// TIA Portal V17 export
// export: Created 2023-12-22T15:04:44.870563Z, ExportSetting WithDefaults, DisplayName Totally Integrated Automation Portal, DisplayVersion V17, DisplayName TIA Portal Openness, DisplayVersion V17, DisplayName TIA Portal Version Control Interface, DisplayVersion V17, DisplayName STEP 7 Professional, DisplayVersion V17, DisplayName STEP 7 Safety, DisplayVersion V17, DisplayName WinCC Advanced, DisplayVersion V17
DATA_BLOCK "tGw_DB"   // DB3
{ S7_Optimized_Access := 'TRUE' }
VERSION : 0.1
// stored: AutoNumber true, DBAccessibleFromOPCUA true, IsOnlyStoredInLoadMemory false, IsRetainMemResEnabled false, IsWriteProtectedInAS false, MemoryReserve 100
   VAR RETAIN
      tGw : Array[0..1] of Struct   // Точка подключения к КП
         IP { S7_SetPoint := 'True'} : IP_V4;
         Port { S7_SetPoint := 'True'} : UInt;
      END_STRUCT;
      "Name" { S7_SetPoint := 'True'} : WString[10] := WSTRING#'1';
      ID { S7_SetPoint := 'True'} : Int := 0;
   END_VAR
BEGIN
   tGw[0].IP.ADDR[1] := 16#0A;
   tGw[0].IP.ADDR[2..3] := 16#01;
   tGw[0].IP.ADDR[4] := 16#9B;
   tGw[1].IP.ADDR[1] := 16#0A;
   tGw[1].IP.ADDR[2..3] := 16#01;
   tGw[1].IP.ADDR[4] := 16#C9;
   tGw[0..1].Port := 503;
END_DATA_BLOCK
